// HMI Banner Structure Relaying Data to HMI Controls
TYPE HMIBanner :
STRUCT
	Text	: T_MaxString;	// Text for HMI Banner
	AltText	: T_MaxString;	// Additional Text for HMI Banner
	Color	: eColor;		// Color of HMI Banner Background
END_STRUCT
END_TYPE

(* stored: Version 1.1.0.1, ProductVersion 3.1.4024.9
   DUT HMIBanner: Id {46001161-f6c9-4e06-8e94-8f25d704f1d9} *)
